ABB RAPID module: TD05Test.mod

MODULE TD05Test_Mod
    !***********************************************************************
    ! Sample .tgs welding program for the ABB prototype (Phase 2/3).
    !
    ! Stands in for a Weld-Planner-generated program. Mirrors the request
    ! call order of the FANUC sample TD05tRJYQd.ls (one capture set with two
    ! captures + one weld; touch-sense family omitted - out of v1 scope).
    !
    ! Naming contract (plan 4.1): file name = PROC name = the program name
    ! the HMI sends ("TD05Test"); TG_Main loads "HOME:/TGS/"+name+".mod" and
    ! late-binds %name%. The MODULE name carries a "_Mod" suffix because
    ! RAPID module names and global routine names share one namespace - a
    ! module named like its own PROC is a semantic error ("name ambiguous").
    ! It calls the TG_* request PROCs and reads the PERS data from
    ! TG_Comms.sys directly - no include mechanism needed (task-wide scope).
    !
    ! Request calls pass the report tool/frame EXPLICITLY per call
    ! (\Tool/\WObj, plan 7.6 style b - this is what the exporter emits).
    ! The DEPRECATED modal alternative (kept in TG_Comms as the back-pocket
    ! fallback) is shown as comments at each former assignment site.
    !
    ! Motion is MoveAbsJ between safe joint poses so it runs on any virtual
    ! controller. Real capture/weld moves in the received frames are shown
    ! as comments where they belong - except the weld-frame demonstration
    ! (search "demonstration"), which does move in wobjTG_Weld on purpose:
    ! the same target before and after TG_ReqWeldFrame, to show the received
    ! frame taking effect.
    !***********************************************************************

    ! Safe joint poses (VC demo only - a real .tgs program carries its own targets)
    LOCAL CONST jointtarget jtHome:=[[0,0,0,0,30,0],[9E9,9E9,9E9,9E9,9E9,9E9]];
    LOCAL CONST jointtarget jtCap1:=[[15,10,-10,0,40,0],[9E9,9E9,9E9,9E9,9E9,9E9]];
    LOCAL CONST jointtarget jtCap2:=[[-15,10,-10,0,40,0],[9E9,9E9,9E9,9E9,9E9,9E9]];

    ! Weld-frame demonstration target. Coordinates are relative to
    ! wobjTG_Weld, so the SAME target resolves to a different Cartesian
    ! position once TG_ReqWeldFrame writes the frame received from the HMI.
    ! Orientation [0,0,1,0] = tool pointing along -z of the work object.
    LOCAL CONST robtarget rtWeldDemo:=[[1000,0,600],[0,0,1,0],[0,0,0,0],[9E9,9E9,9E9,9E9,9E9,9E9]];

    PROC TD05Test()
        ! --- program header (FANUC lines 1-8) ---
        stTG_ProgPass:="TD05Test";     ! SET_PASS_SR: program name == password
        stTG_RobStatus:="Ok";          ! SET_ROB_S_SR('Ok')
        stTG_SubName:="none";          ! deterministic start (SR[25] was stale on FANUC)

        ! --- work objects (weld_frame_update_strategy_v1) ----------------
        ! The program assigns the frame nominals here, before any motion;
        ! the requests below overwrite the .oframe component with the
        ! measured frame. ufprog/ufmec are never written at runtime.
        !
        ! WHY uframe IS RESET TOO, and it is contract rather than tidiness.
        ! The non-coordinated case is correct only BECAUSE uframe is
        ! identity, which makes uframe*oframe = oframe = the frame the HMI
        ! served. That is a claim about the LIVE PERS value, and a PERS
        ! keeps whatever it was last assigned - across loads and across a
        ! saved station. A controller that ever ran the pre-2026-09-03 code,
        ! which served the frame INTO uframe, still holds a frame there;
        ! composing it with the new oframe write double-transforms every
        ! pose silently, while a watch on oframe reads exactly right. So
        ! normalize it at entry. THE WELD PLANNER ABB EXPORTER MUST EMIT
        ! THE SAME RESET for every base-referenced work object its program
        ! uses - .uframe is assumed identity everywhere downstream.
        !
        ! This demo is not coordinated, so the weld uses the
        ! base-referenced wobjTG_Weld. A coordinated weld would pass its
        ! station's object instead - wobjTG_WeldStn1 or wobjTG_WeldStn2,
        ! see TD05Weld.mod - and would NOT reset
        ! uframe: the controller derives that one itself and ignores the
        ! declared value.
        ! The CAMERA object is always wobjTG_Cam, base-referenced, for a
        ! coordinated weld too: captures are standstill captures at one
        ! index, and keeping them base-referenced keeps the HMI's scan and
        ! registration path identical to FANUC's.
        wobjTG_Cam.uframe:=[[0,0,0],[1,0,0,0]];
        wobjTG_Cam.oframe:=[[0,0,0],[1,0,0,0]];
        wobjTG_Weld.uframe:=[[0,0,0],[1,0,0,0]];
        wobjTG_Weld.oframe:=[[0,0,0],[1,0,0,0]];

        ! DEPRECATED modal alternative (plan 7.6): nTG_ActTool:=8; nTG_ActFrame:=0;
        MoveAbsJ jtHome,v100,fine,tTG_Weld;

        ! --- password / dry-run check (FANUC lines 9-16) ---
        ! Torch tool, home frame -> base for the demo (FANUC UT[8]/UFRAME[9])
        TG_ReqPassCheck \Tool:=tTG_Weld \WObj:=wobj0;
        IF nTG_PassOK=0 THEN
            ! FANUC: 'END' - terminate immediately, NO end request (R_E).
            RETURN;
        ENDIF
        ! Dry-run handling (FANUC lines 13-16): default welding ON, then
        ! disable it when the HMI sent dry_run=1. Placeholder PROCs in
        ! TG_Cell.sys - empty until the real cell's weld-enable I/O exists.
        TG_DryRunOff;
        IF nTG_DryRun=1 TG_DryRunOn;
        ! FANUC line 18 has CAM_PREP commented out ("!-- CALL CAM_PREP");
        ! TG_CamPrep exists as a placeholder if a cell ever needs it.
        TG_WeldPrep;                   ! FANUC line 19

        ! --- capture set (FANUC lines 27-62: camera tool UT[2], frame UFRAME[5]) ---
        ! \WObj:=wobjTG_Cam is both the report frame AND the wobj the request
        ! writes the served frame into (through the PERS reference), so the
        ! frame received by TG_ReqCamFrame is used from the very next pose
        ! report (FANUC needed UFRAME[5]=PR[5] re-emits).
        ! DEPRECATED modal alternative (plan 7.6): nTG_ActTool:=2; nTG_ActFrame:=5;
        MoveAbsJ jtCap1,v100,fine,tTG_Cam;
        stTG_SubName:="C1PGlobal_m45_3";
        TG_ReqCamFrame \Tool:=tTG_Cam \WObj:=wobjTG_Cam;   ! R_C_F -> wobjTG_Cam.oframe + nTG_DoCapture
        ! 2 = robot-side abort sentinel: bad frame payload (matrix I4)
        IF nTG_DoCapture=2 GOTO abort_end;
        IF nTG_DoCapture=1 THEN
            TG_CamOpen;                ! FANUC CALL CAM_OPEN
            ! Real program: move to the capture point in the just-received
            ! frame:
            !   MoveJ pCap1,v100,fine,tTG_Cam\WObj:=wobjTG_Cam;
            WaitTime 0.2;              ! FANUC: WAIT 0.20(sec)
            TG_ReqCapture \Tool:=tTG_Cam \WObj:=wobjTG_Cam;   ! R_C -> nTG_CaptureOK
            IF nTG_CaptureOK=0 GOTO abort_end;
        ENDIF
        MoveAbsJ jtCap2,v100,fine,tTG_Cam;
        stTG_SubName:="C2PGlobal_m45_3";
        TG_ReqCamFrame \Tool:=tTG_Cam \WObj:=wobjTG_Cam;
        IF nTG_DoCapture=2 GOTO abort_end;
        IF nTG_DoCapture=1 THEN
            TG_CamOpen;                ! FANUC CALL CAM_OPEN
            WaitTime 0.2;
            TG_ReqCapture \Tool:=tTG_Cam \WObj:=wobjTG_Cam;
            IF nTG_CaptureOK=0 GOTO abort_end;
        ENDIF

        ! --- end of captures: global localization (FANUC lines 61-63) ---
        TG_ReqGlobalCapDone;           ! R_G_C_D -> nTG_GlobalCapOK
        TG_CamClose;                   ! FANUC CALL CAM_CLOSE
        TG_WeldPrep;                   ! FANUC line 63 (before the weld transition)

        ! --- weld (FANUC lines 197-226: torch UT[8], frame UFRAME[6]) ---
        ! DEPRECATED modal alternative (plan 7.6): nTG_ActTool:=8; nTG_ActFrame:=6;
        stTG_SubName:="PWeld2";

        ! ---------------- weld-frame demonstration (demo only) ----------------
        ! Same target, moved to BEFORE and AFTER the frame request. Because
        ! rtWeldDemo is expressed in wobjTG_Weld, the robot ends up in two
        ! different Cartesian positions - visible proof that TG_ReqWeldFrame
        ! updated the frame the welding motions run in.
        !
        ! Back to the identity nominal first, so the "before" position is
        ! the same on every cycle (wobjTG_Weld otherwise persists from the
        ! previous run, exactly like FANUC UFRAME[6] does). uframe needs no
        ! repeat - nothing writes it after the entry normalization above.
        ! DEMO-ONLY, and the distinction is worth being exact about:
        ! assigning the nominal AT ENTRY is prescribed (see the header
        ! block), but a production .tgs must never re-assign a work object
        ! frame MID-RUN, between a TG_ReqWeldFrame and the weld it serves.
        ! That would discard the frame the HMI just served and re-open the
        ! O-3 look-ahead hazard.
        wobjTG_Weld.oframe:=[[0,0,0],[1,0,0,0]];
        ! The same target in two different frames needs two different arm
        ! configurations, so the stored confdata cannot satisfy both.
        ! Demo-only: a production program keeps configuration control on.
        ConfJ\Off;
        ConfL\Off;
        MoveJ rtWeldDemo,v200,fine,tTG_Weld\WObj:=wobjTG_Weld;
        TPWrite "TG DEMO: before R_W_F, TCP ="\Pos:=CPos(\Tool:=tTG_Weld \WObj:=wobj0);
        ! ----------------------------------------------------------------------

        TG_ReqWeldFrame \Tool:=tTG_Weld \WObj:=wobjTG_Weld;   ! R_W_F -> wobjTG_Weld.oframe + nTG_WeldStatus
        TG_CamClose;                   ! FANUC defensive CAM_CLOSE after R_W_F
        IF nTG_WeldStatus=2 GOTO abort_end;
        IF nTG_WeldStatus=1 THEN
            ! ------------- weld-frame demonstration, part 2 -------------
            ! Identical instruction, identical target - new frame.
            MoveJ rtWeldDemo,v200,fine,tTG_Weld\WObj:=wobjTG_Weld;
            TPWrite "TG DEMO: after  R_W_F, TCP ="\Pos:=CPos(\Tool:=tTG_Weld \WObj:=wobj0);
            ! -----------------------------------------------------------
            ! Approach in the received weld frame:
            !   MoveJ pApproach,v100,z100,tTG_Weld\WObj:=wobjTG_Weld;
            !   MoveL pWeldStart,v50,fine,tTG_Weld\WObj:=wobjTG_Weld;
            TG_ReqWeldParams;          ! R_W_P -> nTG_UdwpFlag, nTG_TravelSpeed, ...
            ! RobotWare Arc weld goes here (plan, phase 4): ArcLStart/ArcL/
            ! ArcLEnd with welddata built from nTG_WeldProc/nTG_WireFeed/
            ! nTG_ArcLength/nTG_ArcControl, travel speed nTG_TravelSpeed
            ! (FANUC: L P[124] R[175]inch/min + WELD START/END[R[171],20]).
            ! This program has no Arc option, so no weld actually runs here.

            ! R_W_S (FANUC: CALL R_W_S right after WELD END). DUMMY stats -
            ! this module cannot weld, so there is nothing real to measure;
            ! the fixed values below make the request assertable in a
            ! transcript. succ_ae follows the dry-run flag exactly as a real
            ! weld would: welding inhibited -> no arc -> the HMI must NOT
            ! record an analytics row.
            nTG_WeldDist:=123.456;
            nTG_ArcOnTime:=7.89;
            nTG_SuccArcEnd:=1-nTG_DryRun;
            TG_ReqWeldStats;           ! R_W_S -> "dist,arc_on,succ_ae"
        ENDIF

        ! --- return home (FANUC lines 397-411) ---
        TG_CamClose;                   ! FANUC CALL CAM_CLOSE
        MoveAbsJ jtHome,v100,fine,tTG_Weld;

abort_end:
        ! FANUC LBL[101]: both the normal exit and the abort target.
        ! R_E's pose is reported in torch/weld frame regardless of which
        ! section aborted (a shared label cannot know; the modal version
        ! reported whatever was last selected). Safe: the HMI ignores every
        ! R_E pose (plan 1.4.1). Matches the modal version on the normal
        ! path, so transcripts stay comparable.
        ConfJ\On;                      ! undo the demo's relaxed config control
        ConfL\On;
        stTG_SubName:="none";
        TG_ReqEnd \Tool:=tTG_Weld \WObj:=wobjTG_Weld;   ! R_E
    ENDPROC

ENDMODULE
